// TIA Portal V17 program export: 1 tag tables, 0 data types, 0 data blocks, 2 code blocks (in call order from the OBs), 0 instance data blocks

VAR_GLOBAL   // PLC tag table "Default tag table"
   alwaysTrue AT %M0.0 : Bool;
   alwaysFalse AT %M1.0 : Bool;
   Tag_1 AT %MW10 : Int;
END_VAR

ORGANIZATION_BLOCK "Main"   // OB1, LAD, ProgramCycle
TITLE = "Main Program Sweep (Cycle)"
{ S7_Optimized_Access := 'TRUE' }
VERSION : 0.1
// stored: AutoNumber true, IsIECCheckEnabled false, SetENOAutomatically false
   VAR_INPUT
      Initial_Call : Bool;   // Initial call of this OB
      Remanence : Bool;   // =True, if remanent data are available
   END_VAR
BEGIN

REGION Network 1
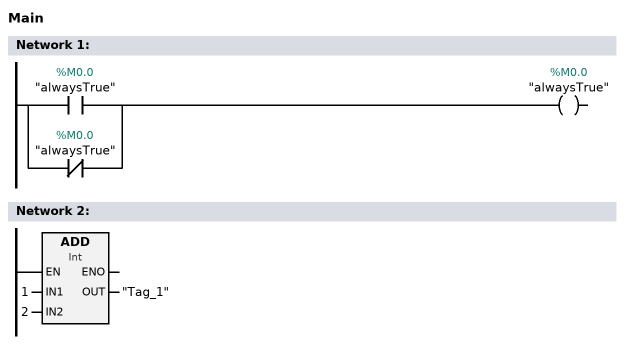
   RUNG wire#powerrail
      Contact( "alwaysTrue" )
      wire#w1
      Coil( "alwaysTrue" )
   END_RUNG
   RUNG wire#powerrail
      I_Contact( "alwaysTrue" )
   END_RUNG wire#w1
   // the same network as SCL:
   "alwaysTrue" := "alwaysTrue" OR NOT "alwaysTrue";
END_REGION

REGION Network 2
   RUNG wire#powerrail
      { S7_Templates := "SrcType := Int" } Add(in1 := 1, in2 := 2, out => "Tag_1")
   END_RUNG
   // the same network as SCL:
   "Tag_1" := 1 + 2;
END_REGION
END_ORGANIZATION_BLOCK

FUNCTION "Block_1" : Void   // FC1, LAD
{ S7_Optimized_Access := 'TRUE' }
VERSION : 0.1
// stored: AutoNumber true, IsIECCheckEnabled false, SetENOAutomatically false, UDAEnableTagReadback false
BEGIN

REGION Network 2
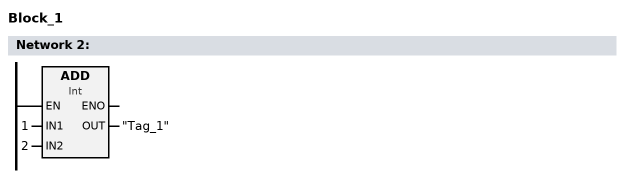
   RUNG wire#powerrail
      { S7_Templates := "SrcType := Int" } Add(in1 := 1, in2 := 2, out => "Tag_1")
   END_RUNG
   // the same network as SCL:
   "Tag_1" := 1 + 2;
END_REGION
END_FUNCTION
